(* LS Electric XG5000 project: 241004_실습6_푸시버튼으로토글기능구현 *)
(* PLC LSPLC *)

PROGRAM NewProgram (* task: 스캔 프로그램 *)
VAR
    내부메모리1 AT %MX0 : BOOL; (* 양변환 토글 동작 *)
    내부메모리2 AT %MX1 : BOOL; (* 음변환 토글 동작 *)
    내부메모리3 AT %MX2 : BOOL; (* 토글 동작, 자기유지 *)
    녹색램프 AT %QX0.1.0 : BOOL; (* 토글 스위치, 녹색램프 *)
    푸시버튼1 AT %IX0.0.0 : BOOL; (* 양변환 검출 푸시버튼 스위치 *)
END_VAR
VAR
    _e1 : R_TRIG;
    _e2 : R_TRIG;
    _e3 : F_TRIG;
    _e4 : F_TRIG;
    _e5 : R_TRIG;
    _e6 : R_TRIG;
END_VAR

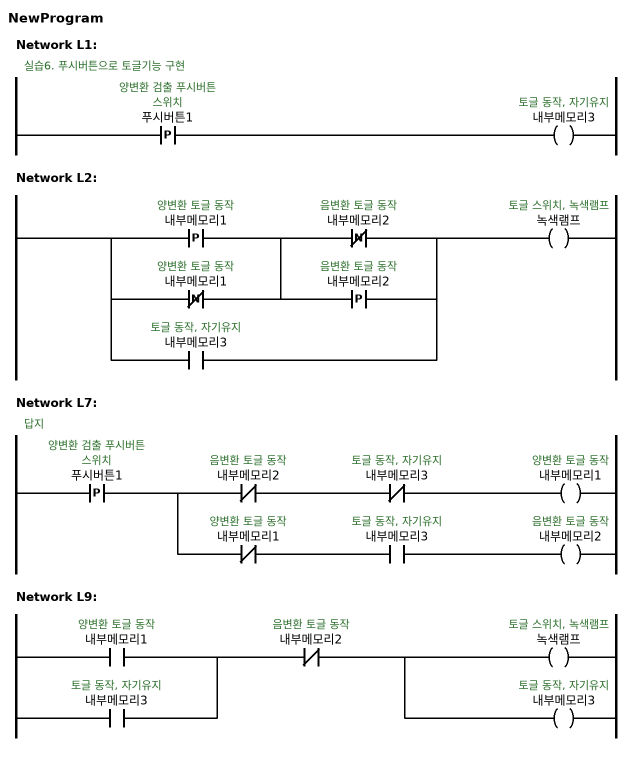
(* 실습6. 푸시버튼으로 토글기능 구현 *)
(* Rung L1 *)
_e1(CLK := 푸시버튼1);
내부메모리3 := _e1.Q;
(* Rung L2 *)
_e2(CLK := 내부메모리1);
_e3(CLK := 내부메모리1);
_e4(CLK := 내부메모리2);
_e5(CLK := 내부메모리2);
녹색램프 := ((_e2.Q OR NOT _e3.Q) AND (NOT _e4.Q OR _e5.Q)) OR 내부메모리3;
(* 답지 *)
(* Rung L7 *)
_e6(CLK := 푸시버튼1);
내부메모리1 := _e6.Q AND NOT 내부메모리2 AND NOT 내부메모리3;
내부메모리2 := _e6.Q AND NOT 내부메모리1 AND 내부메모리3;
(* Rung L9 *)
녹색램프 := (내부메모리1 OR 내부메모리3) AND NOT 내부메모리2;
내부메모리3 := (내부메모리1 OR 내부메모리3) AND NOT 내부메모리2;
END_PROGRAM